// TIA Portal V19 export
TYPE "typeSimSensors"
   STRUCT
      Sensors : Struct
         Sensor11 : Real;   // Machine 001 / Sensor 001
         Sensor12 : Real;   // Machine 001 / Sensor 002
         Sensor13 : Real;   // Machine 001 / Sensor 003
         Sensor14 : Real;   // Machine 001 / Sensor 004
         Sensor21 : Real;   // Machine 002 / Sensor 001
         Sensor22 : Real;   // Machine 002 / Sensor 002
         Sensor23 : Real;   // Machine 002 / Sensor 003
         Sensor24 : Real;   // Machine 002 / Sensor 004
      END_STRUCT;
   END_STRUCT;
END_TYPE
